{attribute 'GeneratedUsingTerminal: EL6851-0010-0016'}
{attribute addProperty BoxType "EL6851-0010-0016"}
{attribute addProperty Id "ChannelAT %I*ARRAY[0..63] OF USINT64"}
{attribute addProperty CRC "2289174522"}
{attribute addProperty Size "64"}
TYPE DMX_Channel_005FDEFD :
STRUCT
	{attribute addProperty Name "Channel"}
	Channel AT %I* : ARRAY[0..63] OF USINT;
END_STRUCT
END_TYPE

(* stored: Version 1.2.0.0, ProductVersion 3.1.4024.9
   DUT DMX_Channel_005FDEFD: Id {4d6147b7-4dc8-4e79-a6bc-3c510193f9b6} *)
